// TIA Portal project "LONGHAI_V15.1" (V15.1)

(* hardware
DEVICE "S7-1200 station_1"  S7-1200 Station
   slot 0: "Rack_0"  S7-1200 Rack  Rack  V1.0
   slot 1: "PLC_1"  CPU 1211C DC/DC/DC  6ES7 211-1AE40-0XB0  V4.2
*)

// ===== PLC "PLC_1"  CPU 1211C DC/DC/DC =====

VAR_GLOBAL   // PLC tag table "Default tag table"
   "Sensor" AT %I0.2 : Bool;
   "PulseEncoder" AT %ID1000 : DInt;
   "CTXilanh1" AT %I0.3 : Bool;
   "CTXilanh2" AT %I0.4 : Bool;
   "ResetSTT2Xilanh" AT %I0.5 : Bool;
   "Xilanh1" AT %Q0.0 : Bool;
   "Xilanh2" AT %Q0.1 : Bool;
   "Alarm_1" AT %Q0.2 : Bool;
   "Alarm_2" AT %Q0.3 : Bool;
   "SetPulse_Xilanh1_1" AT %MD5 : DInt;
   "WidthFulse" AT %MD50 : Time;
   "OnOffXilanh1" AT %M0.0 : Bool;
   "OnOffXilanh2" AT %M0.1 : Bool;
   "ResetSW" AT %M0.5 : Bool;
   "KichReset" AT %M0.3 : Bool;
   "SetPulse_Xilanh1_2" AT %MD70 : DInt;
   "SetPulse_Xilanh2" AT %MD100 : Time;
END_VAR

// folder: System blocks/Program resources

DATA_BLOCK "IEC_Timer_0_DB"   // DB2
{ S7_Optimized_Access := 'TRUE' }
AUTHOR : Simatic
FAMILY : IEC
NAME : IEC_TMR
VERSION : 1.0
// stored: InstanceOfName IEC_TIMER
"IEC_TIMER"
BEGIN
END_DATA_BLOCK

DATA_BLOCK "IEC_Timer_0_DB_1"   // DB3
{ S7_Optimized_Access := 'TRUE' }
AUTHOR : Simatic
FAMILY : IEC
NAME : IEC_TMR
VERSION : 1.0
// stored: InstanceOfName IEC_TIMER
"IEC_TIMER"
BEGIN
END_DATA_BLOCK

DATA_BLOCK "IEC_Timer_0_DB_2"   // DB4
{ S7_Optimized_Access := 'TRUE' }
AUTHOR : Simatic
FAMILY : IEC
NAME : IEC_TMR
VERSION : 1.0
// stored: InstanceOfName IEC_TIMER
"IEC_TIMER"
BEGIN
END_DATA_BLOCK

DATA_BLOCK "IEC_Timer_0_DB_3"   // DB5
{ S7_Optimized_Access := 'TRUE' }
AUTHOR : Simatic
FAMILY : IEC
NAME : IEC_TMR
VERSION : 1.0
// stored: InstanceOfName IEC_TIMER
"IEC_TIMER"
BEGIN
END_DATA_BLOCK

// folder: (top level)

ORGANIZATION_BLOCK "Main"   // OB1, LAD, ProgramCycle
TITLE = "Main Program Sweep (Cycle)"
{ S7_Optimized_Access := 'TRUE' }
VERSION : 0.1
   VAR_INPUT
      Initial_Call : Bool;   // Initial call of this OB
      Remanence : Bool;   // =True, if remanent data are available
   END_VAR
BEGIN

REGION Network 1: Xilanh1
   // đóng xilanh 1
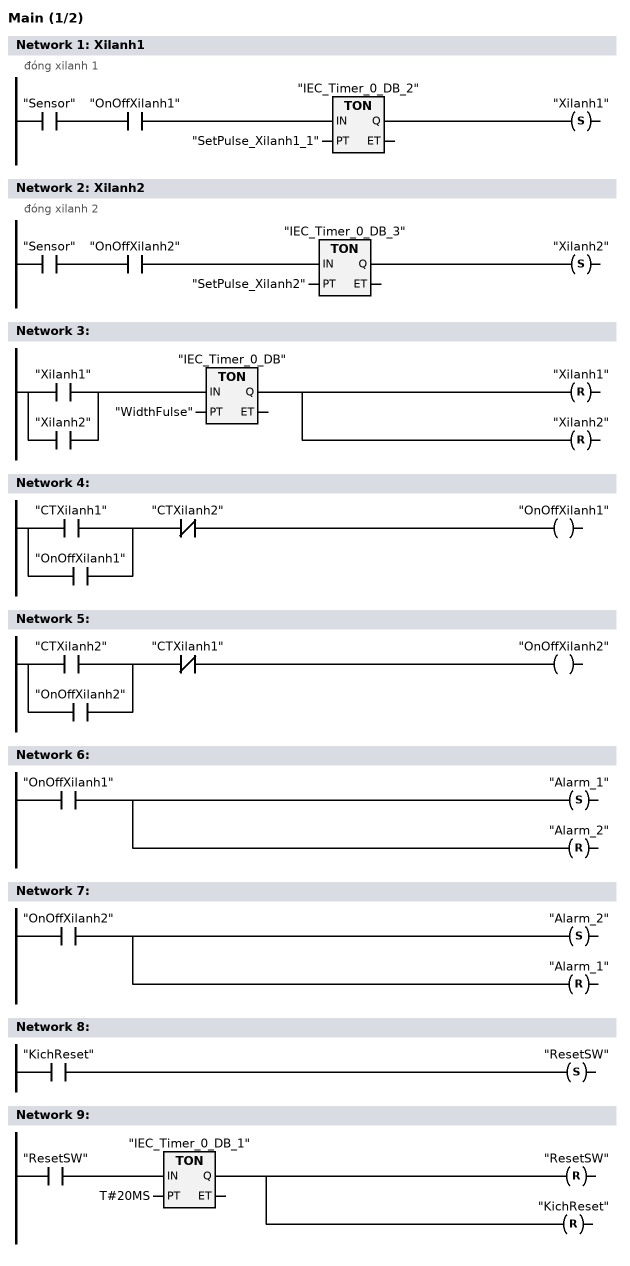
   "IEC_Timer_0_DB_2".TON(IN := "Sensor" AND "OnOffXilanh1", PT := "SetPulse_Xilanh1_1");
   IF "IEC_Timer_0_DB_2".Q THEN "Xilanh1" := TRUE; END_IF;
END_REGION

REGION Network 2: Xilanh2
   // đóng xilanh 2
   "IEC_Timer_0_DB_3".TON(IN := "Sensor" AND "OnOffXilanh2", PT := "SetPulse_Xilanh2");
   IF "IEC_Timer_0_DB_3".Q THEN "Xilanh2" := TRUE; END_IF;
END_REGION

REGION Network 3
   "IEC_Timer_0_DB".TON(IN := "Xilanh1" OR "Xilanh2", PT := "WidthFulse");
   IF "IEC_Timer_0_DB".Q THEN
       "Xilanh1" := FALSE;
       "Xilanh2" := FALSE;
   END_IF;
END_REGION

REGION Network 4
   RUNG wire#powerrail
      Contact( "CTXilanh1" )
      wire#w1
      I_Contact( "CTXilanh2" )
      Coil( "OnOffXilanh1" )
   END_RUNG
   RUNG wire#powerrail
      Contact( "OnOffXilanh1" )
   END_RUNG wire#w1
   // the same network as SCL:
   "OnOffXilanh1" := ("CTXilanh1" OR "OnOffXilanh1") AND NOT "CTXilanh2";
END_REGION

REGION Network 5
   RUNG wire#powerrail
      Contact( "CTXilanh2" )
      wire#w1
      I_Contact( "CTXilanh1" )
      Coil( "OnOffXilanh2" )
   END_RUNG
   RUNG wire#powerrail
      Contact( "OnOffXilanh2" )
   END_RUNG wire#w1
   // the same network as SCL:
   "OnOffXilanh2" := ("CTXilanh2" OR "OnOffXilanh2") AND NOT "CTXilanh1";
END_REGION

REGION Network 6
   RUNG wire#powerrail
      Contact( "OnOffXilanh1" )
      wire#w1
      S_Coil( "Alarm_1" )
   END_RUNG
   RUNG wire#w1
      R_Coil( "Alarm_2" )
   END_RUNG
   // the same network as SCL:
   IF "OnOffXilanh1" THEN
       "Alarm_1" := TRUE;
       "Alarm_2" := FALSE;
   END_IF;
END_REGION

REGION Network 7
   RUNG wire#powerrail
      Contact( "OnOffXilanh2" )
      wire#w1
      S_Coil( "Alarm_2" )
   END_RUNG
   RUNG wire#w1
      R_Coil( "Alarm_1" )
   END_RUNG
   // the same network as SCL:
   IF "OnOffXilanh2" THEN
       "Alarm_2" := TRUE;
       "Alarm_1" := FALSE;
   END_IF;
END_REGION

REGION Network 8
   RUNG wire#powerrail
      Contact( "KichReset" )
      S_Coil( "ResetSW" )
   END_RUNG
   // the same network as SCL:
   IF "KichReset" THEN "ResetSW" := TRUE; END_IF;
END_REGION

REGION Network 9
   "IEC_Timer_0_DB_1".TON(IN := "ResetSW", PT := T#20MS);
   IF "IEC_Timer_0_DB_1".Q THEN
       "ResetSW" := FALSE;
       "KichReset" := FALSE;
   END_IF;
END_REGION

REGION Network 10
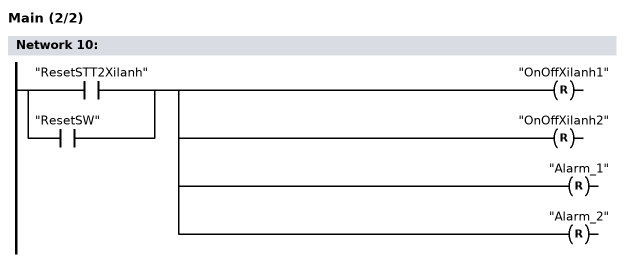
   RUNG wire#powerrail
      Contact( "ResetSTT2Xilanh" )
      wire#w1
      R_Coil( "OnOffXilanh1" )
   END_RUNG
   RUNG wire#powerrail
      Contact( "ResetSW" )
   END_RUNG wire#w1
   RUNG wire#w1
      R_Coil( "OnOffXilanh2" )
   END_RUNG
   RUNG wire#w1
      R_Coil( "Alarm_1" )
   END_RUNG
   RUNG wire#w1
      R_Coil( "Alarm_2" )
   END_RUNG
   // the same network as SCL:
   IF "ResetSTT2Xilanh" OR "ResetSW" THEN
       "OnOffXilanh1" := FALSE;
       "OnOffXilanh2" := FALSE;
       "Alarm_1" := FALSE;
       "Alarm_2" := FALSE;
   END_IF;
END_REGION
END_ORGANIZATION_BLOCK